(* Logix 5000 project; controller NSH_PLC1 vendor 1 type 14 code 167 rev 32.11; software revision 32.02; part 7 of 12 *)
(* tags used below, declared in another part *)
   TempMotor : Motor;   // Temp Motor Tag for Subroutines
   H32D : Motor;   // Shr.Roll.
   H33A : Motor;   // Aspirator
   H34A : Motor;   // HC Vib.
   H34B : Motor;   // Hard Crkr.
   H34C : Motor;   // S.Roll
   H34D : Motor;   // Shr.Roll.
   H35A : Motor;   // Aspirator
   H35B : Motor;   // Aspirator
   H42A : Motor;   // HC Vib.
   H42B : Motor;   // Hard Crkr.
   H42C : Motor;   // S.Roll
   H42D : Motor;   // Shr.Roll.
   H43A : Motor;   // Aspirator
   H43B : Motor;   // Aspirator
   H44A : Motor;   // HC Vib.
   H44B : Motor;   // Hard Crkr.
   H44C : Motor;   // S.Roll
   H44D : Motor;   // Shr.Roll.
   H45A : Motor;   // Aspirator
   H45B : Motor;   // Aspirator
   H49 : Motor;   // Ele.
   H50A : Motor;   // Auger
   H50B : Motor;   // Auger
   M10 : Motor;   // Vib.
   M10A : Motor;   // Asp.
   M10B : Motor;   // Asp.
   M11 : Motor;   // Ele.
   M16 : Motor;   // Evo.
   M17 : Motor;   // Evo.
   M18 : Motor;   // Vib.
   M19 : Motor;   // Ele.
   M1A : Motor;   // Vib.
   M2 : Motor;   // Vib.
   M27 : Motor;   // Belt
   M28 : Motor;   // Belt
   M29 : Motor;   // Ele.
   M3 : Motor;   // Belt
   M30A : Motor;   // HC Vib.
   M30B : Motor;   // Hard Crkr.
   M30C : Motor;   // Shr.Roll.
   M30D : Motor;   // Shr.Roll.
   M31A : Motor;   // Asp.
   M31B : Motor;   // Asp.
   M32A : Motor;   // Vib.Scrn.
   M32B : Motor;   // Ele.
   M37 : Motor;   // 5x12
   M38A : Motor;   // Asp.
   M38B : Motor;   // Asp.
   M39 : Motor;   // Ele.
   M4 : Motor;   // Vib.
   M40A : Motor;   // Sep.
   M40B : Motor;   // Syn.Fer.
   M41 : Motor;   // Ele.
   M44A : Motor;   // Belt
   M44B : Motor;   // Belt
   M5 : Motor;   // Vib.
   M6 : Motor;   // Belt
   M7 : Motor;   // Ele.
   M8 : Motor;   // Shkr.
   M9A : Motor;   // Asp.
   M9B : Motor;   // Asp.
   S1 : Motor;   // Vib.
   S10 : Motor;   // Auger
   S13 : Motor;   // Ele.
   S14 : Motor;   // Auger
   S15 : Motor;   // Auger
   S16A : Motor;   // Auger
   S16B : Motor;   // Auger
   S17A : Motor;   // HS Cracker
   S17B : Motor;   // Hard Crkr.
   S17C : Motor;   // Shr.Roll.
   S17D : Motor;   // S.Roll
   S18A : Motor;   // HC Vib.
   S18B : Motor;   // Hard Crkr.
   S18C : Motor;   // Shr.Roll.
   S18D : Motor;   // S.Roll
   S19 : Motor;   // Gry.
   S2 : Motor;   // Ele.
   S20 : Motor;   // Ele.
   S21 : Motor;   // Roll Fdr.
   S22A : Motor;   // HC Vib.
   S22B : Motor;   // Hard Crkr.
   S22C : Motor;   // Shr.Roll.
   S22D : Motor;   // S.Roll
   S23A : Motor;   // HC Vib.
   S23B : Motor;   // Hard Crkr.
   S23C : Motor;   // Shr.Roll.
   S23D : Motor;   // S.Roll
   S24 : Motor;   // Deck
   S25 : Motor;   // Ele.
   S26 : Motor;   // Auger
   S27 : Motor;   // Roll Fdr
   S28A : Motor;   // HC Vib.
   S28B : Motor;   // Hard Crkr.
   S28C : Motor;   // Shr.Roll.
   S28D : Motor;   // S.Roll
   S29A : Motor;   // HC Vib.
   S29B : Motor;   // Hard Crkr.
   S29C : Motor;   // Shr.Roll.
   S29D : Motor;   // S.Roll
   S3 : Motor;   // Auger
   S30 : Motor;   // Ele.
   S31 : Motor;   // Auger
   S32A : Motor;   // HC Vib.
   S32B : Motor;   // Hard Crkr.
   S32C : Motor;   // Shr.Roll.
   S32D : Motor;   // S.Roll
   S33A : Motor;   // HC Vib.
   S33B : Motor;   // Hard Crkr.
   S33C : Motor;   // Shr.Roll.
   S33D : Motor;   // S.Roll
   S34 : Motor;   // Deck
   S35 : Motor;   // Ele.
   S36 : Motor;   // Auger
   S37A : Motor;   // HC Vib.
   S37B : Motor;   // Hard Crkr.
   S37C : Motor;   // Shr.Roll.
   S37D : Motor;   // S.Roll
   S38 : Motor;   // Shkr.
   S39 : Motor;   // Ele.
   S40A : Motor;   // HC Vib.
   S40B : Motor;   // Hard Crkr.
   S40C : Motor;   // Shr.Roll.
   S40D : Motor;   // S.Roll
   S41 : Motor;   // Ele.
   S42A : Motor;   // HC Vib.
   S42B : Motor;   // Hard Crkr.
   S42C : Motor;   // S.Roll
   S42D : Motor;   // Shr.Roll.
   S43 : Motor;   // Shkr.
   S44 : Motor;   // Ele.
   S45 : Motor;   // Auger
   S46A : Motor;   // HC Vib.
   S46B : Motor;   // Hard Crkr.
   S46C : Motor;   // S.Roll
   S46D : Motor;   // Shr.Roll.
   S4A : Motor;   // Aspirator
   S4B : Motor;   // Aspirator
   S5A : Motor;   // Aspirator
   S5B : Motor;   // Aspirator
   S6 : Motor;   // Belt
   S7 : Motor;   // Ele.
   S8 : Motor;   // Auger
   S9 : Motor;   // Ele.
(* HullerSheller, continued *)

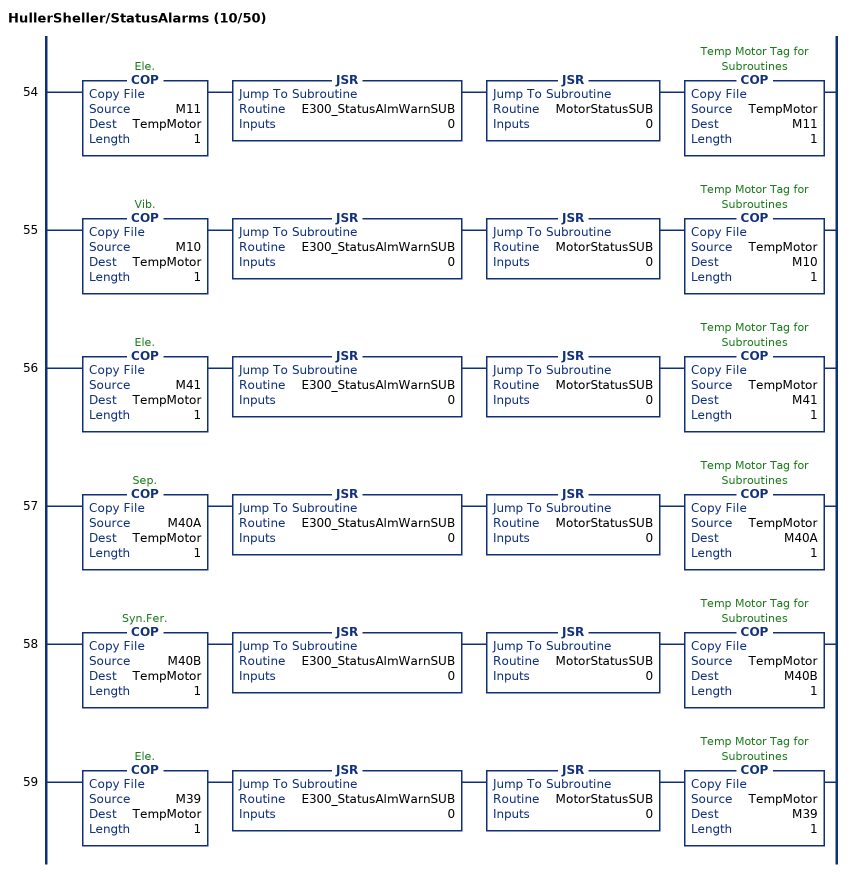
   [picture p138: HullerSheller/StatusAlarms rungs 54-59]
   54: COP(M11,TempMotor,1)JSR(E300_StatusAlmWarnSUB,0)JSR(MotorStatusSUB,0)COP(TempMotor,M11,1);
   55: COP(M10,TempMotor,1)JSR(E300_StatusAlmWarnSUB,0)JSR(MotorStatusSUB,0)COP(TempMotor,M10,1);
   56: COP(M41,TempMotor,1)JSR(E300_StatusAlmWarnSUB,0)JSR(MotorStatusSUB,0)COP(TempMotor,M41,1);
   57: COP(M40A,TempMotor,1)JSR(E300_StatusAlmWarnSUB,0)JSR(MotorStatusSUB,0)COP(TempMotor,M40A,1);
   58: COP(M40B,TempMotor,1)JSR(E300_StatusAlmWarnSUB,0)JSR(MotorStatusSUB,0)COP(TempMotor,M40B,1);
   59: COP(M39,TempMotor,1)JSR(E300_StatusAlmWarnSUB,0)JSR(MotorStatusSUB,0)COP(TempMotor,M39,1);
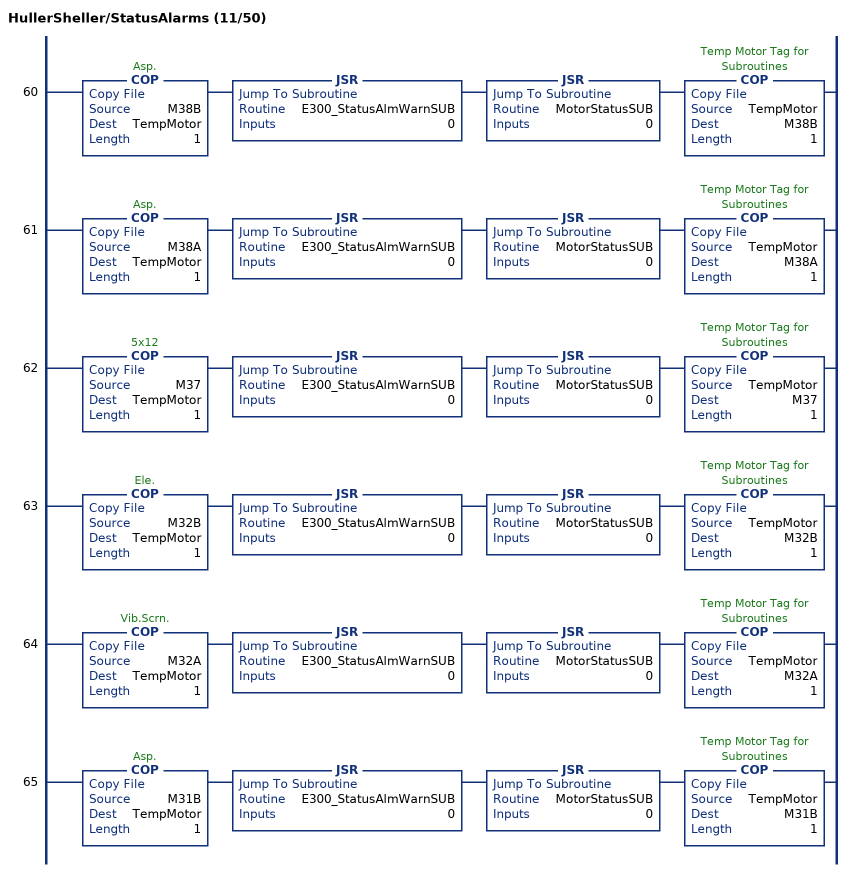
   60: COP(M38B,TempMotor,1)JSR(E300_StatusAlmWarnSUB,0)JSR(MotorStatusSUB,0)COP(TempMotor,M38B,1);
   61: COP(M38A,TempMotor,1)JSR(E300_StatusAlmWarnSUB,0)JSR(MotorStatusSUB,0)COP(TempMotor,M38A,1);
   62: COP(M37,TempMotor,1)JSR(E300_StatusAlmWarnSUB,0)JSR(MotorStatusSUB,0)COP(TempMotor,M37,1);
   63: COP(M32B,TempMotor,1)JSR(E300_StatusAlmWarnSUB,0)JSR(MotorStatusSUB,0)COP(TempMotor,M32B,1);
   64: COP(M32A,TempMotor,1)JSR(E300_StatusAlmWarnSUB,0)JSR(MotorStatusSUB,0)COP(TempMotor,M32A,1);
   65: COP(M31B,TempMotor,1)JSR(E300_StatusAlmWarnSUB,0)JSR(MotorStatusSUB,0)COP(TempMotor,M31B,1);
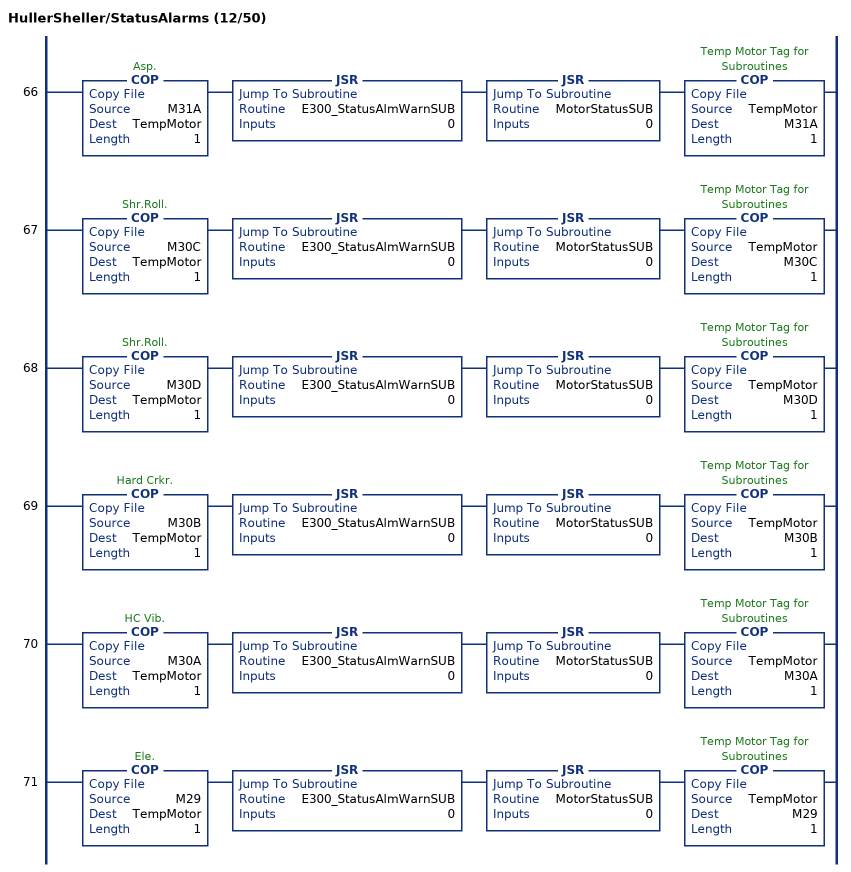
   66: COP(M31A,TempMotor,1)JSR(E300_StatusAlmWarnSUB,0)JSR(MotorStatusSUB,0)COP(TempMotor,M31A,1);
   67: COP(M30C,TempMotor,1)JSR(E300_StatusAlmWarnSUB,0)JSR(MotorStatusSUB,0)COP(TempMotor,M30C,1);
   68: COP(M30D,TempMotor,1)JSR(E300_StatusAlmWarnSUB,0)JSR(MotorStatusSUB,0)COP(TempMotor,M30D,1);
   69: COP(M30B,TempMotor,1)JSR(E300_StatusAlmWarnSUB,0)JSR(MotorStatusSUB,0)COP(TempMotor,M30B,1);
   70: COP(M30A,TempMotor,1)JSR(E300_StatusAlmWarnSUB,0)JSR(MotorStatusSUB,0)COP(TempMotor,M30A,1);
   71: COP(M29,TempMotor,1)JSR(E300_StatusAlmWarnSUB,0)JSR(MotorStatusSUB,0)COP(TempMotor,M29,1);
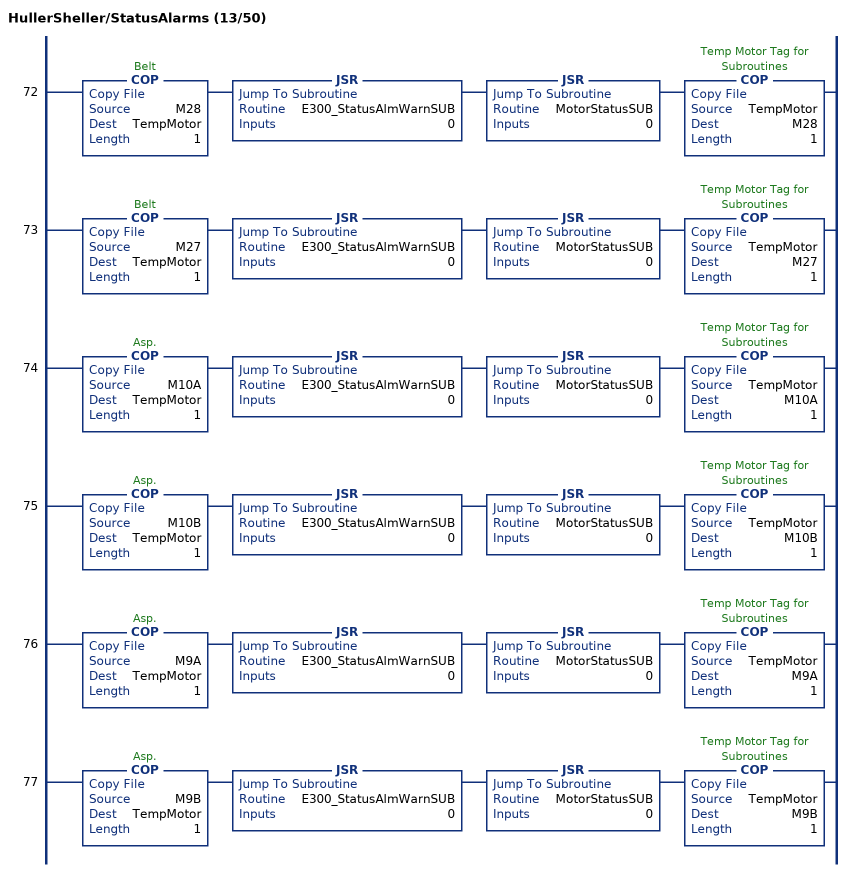
   72: COP(M28,TempMotor,1)JSR(E300_StatusAlmWarnSUB,0)JSR(MotorStatusSUB,0)COP(TempMotor,M28,1);
   73: COP(M27,TempMotor,1)JSR(E300_StatusAlmWarnSUB,0)JSR(MotorStatusSUB,0)COP(TempMotor,M27,1);
   74: COP(M10A,TempMotor,1)JSR(E300_StatusAlmWarnSUB,0)JSR(MotorStatusSUB,0)COP(TempMotor,M10A,1);
   75: COP(M10B,TempMotor,1)JSR(E300_StatusAlmWarnSUB,0)JSR(MotorStatusSUB,0)COP(TempMotor,M10B,1);
   76: COP(M9A,TempMotor,1)JSR(E300_StatusAlmWarnSUB,0)JSR(MotorStatusSUB,0)COP(TempMotor,M9A,1);
   77: COP(M9B,TempMotor,1)JSR(E300_StatusAlmWarnSUB,0)JSR(MotorStatusSUB,0)COP(TempMotor,M9B,1);
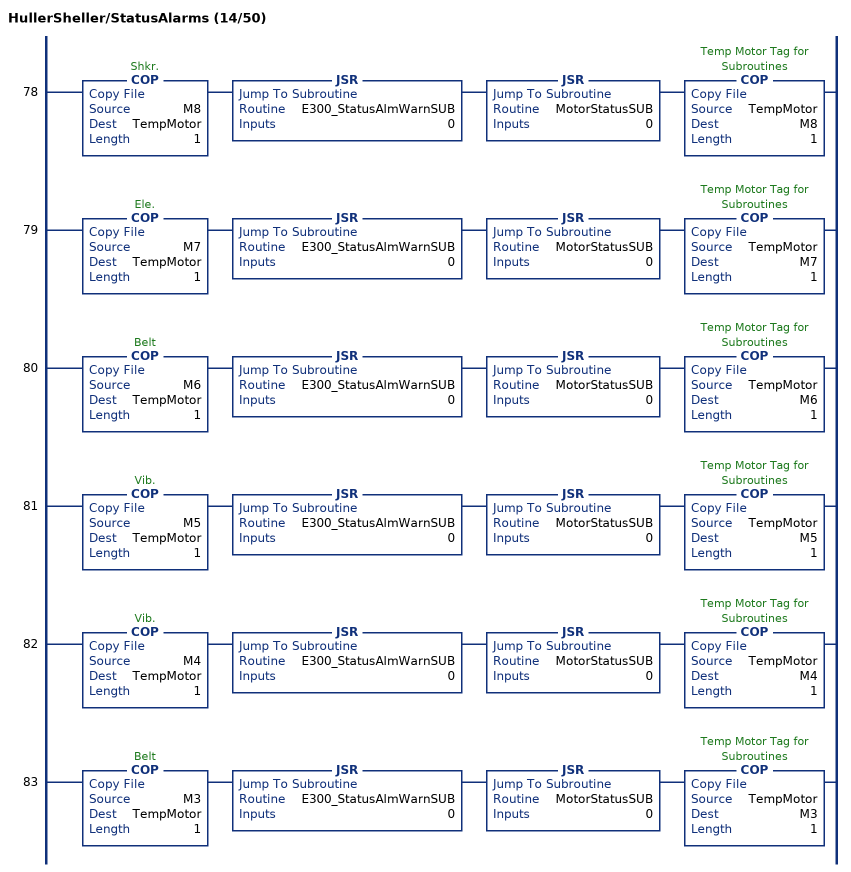
   78: COP(M8,TempMotor,1)JSR(E300_StatusAlmWarnSUB,0)JSR(MotorStatusSUB,0)COP(TempMotor,M8,1);
   79: COP(M7,TempMotor,1)JSR(E300_StatusAlmWarnSUB,0)JSR(MotorStatusSUB,0)COP(TempMotor,M7,1);
   80: COP(M6,TempMotor,1)JSR(E300_StatusAlmWarnSUB,0)JSR(MotorStatusSUB,0)COP(TempMotor,M6,1);
   81: COP(M5,TempMotor,1)JSR(E300_StatusAlmWarnSUB,0)JSR(MotorStatusSUB,0)COP(TempMotor,M5,1);
   82: COP(M4,TempMotor,1)JSR(E300_StatusAlmWarnSUB,0)JSR(MotorStatusSUB,0)COP(TempMotor,M4,1);
   83: COP(M3,TempMotor,1)JSR(E300_StatusAlmWarnSUB,0)JSR(MotorStatusSUB,0)COP(TempMotor,M3,1);
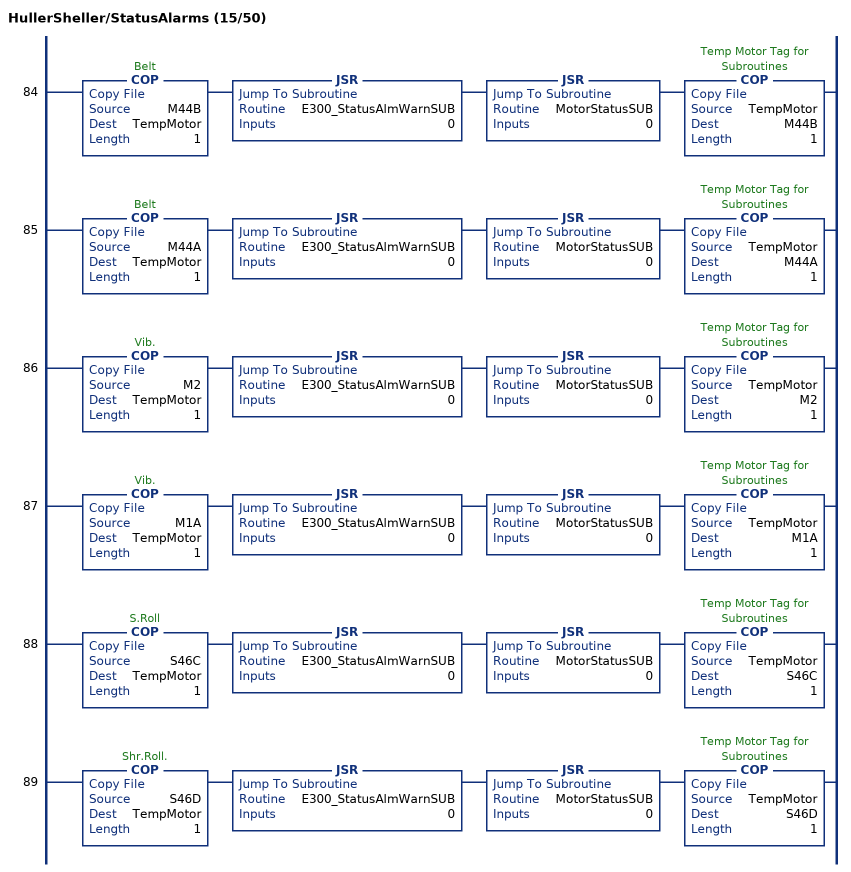
   84: COP(M44B,TempMotor,1)JSR(E300_StatusAlmWarnSUB,0)JSR(MotorStatusSUB,0)COP(TempMotor,M44B,1);
   85: COP(M44A,TempMotor,1)JSR(E300_StatusAlmWarnSUB,0)JSR(MotorStatusSUB,0)COP(TempMotor,M44A,1);
   86: COP(M2,TempMotor,1)JSR(E300_StatusAlmWarnSUB,0)JSR(MotorStatusSUB,0)COP(TempMotor,M2,1);
   87: COP(M1A,TempMotor,1)JSR(E300_StatusAlmWarnSUB,0)JSR(MotorStatusSUB,0)COP(TempMotor,M1A,1);
   88: COP(S46C,TempMotor,1)JSR(E300_StatusAlmWarnSUB,0)JSR(MotorStatusSUB,0)COP(TempMotor,S46C,1);
   89: COP(S46D,TempMotor,1)JSR(E300_StatusAlmWarnSUB,0)JSR(MotorStatusSUB,0)COP(TempMotor,S46D,1);
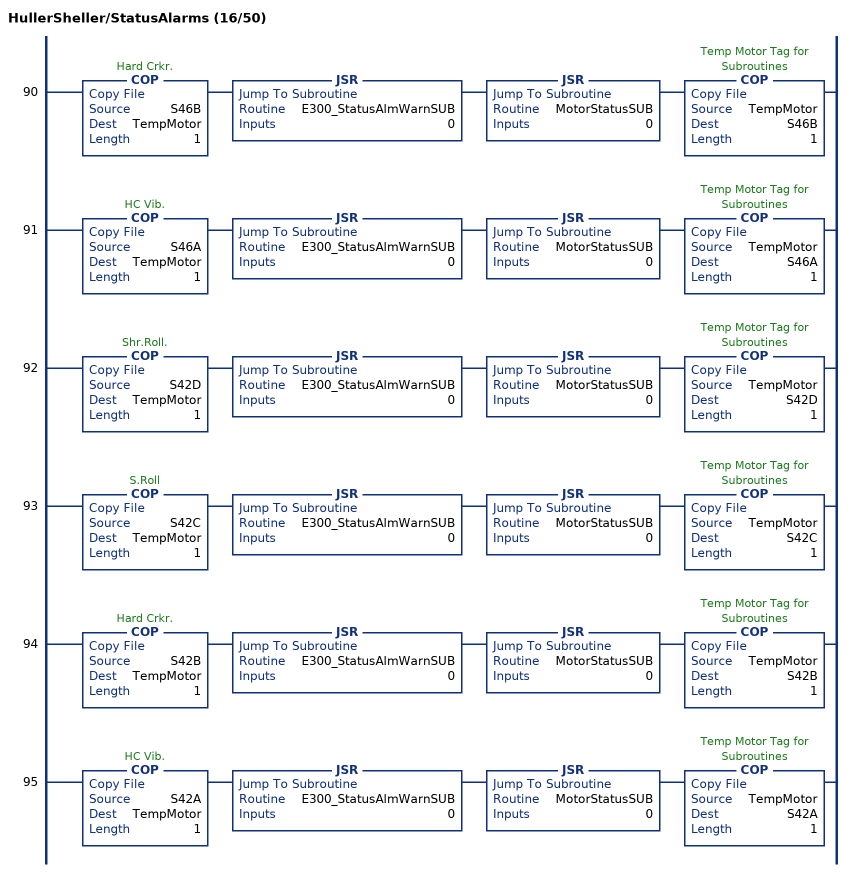
   90: COP(S46B,TempMotor,1)JSR(E300_StatusAlmWarnSUB,0)JSR(MotorStatusSUB,0)COP(TempMotor,S46B,1);
   91: COP(S46A,TempMotor,1)JSR(E300_StatusAlmWarnSUB,0)JSR(MotorStatusSUB,0)COP(TempMotor,S46A,1);
   92: COP(S42D,TempMotor,1)JSR(E300_StatusAlmWarnSUB,0)JSR(MotorStatusSUB,0)COP(TempMotor,S42D,1);
   93: COP(S42C,TempMotor,1)JSR(E300_StatusAlmWarnSUB,0)JSR(MotorStatusSUB,0)COP(TempMotor,S42C,1);
   94: COP(S42B,TempMotor,1)JSR(E300_StatusAlmWarnSUB,0)JSR(MotorStatusSUB,0)COP(TempMotor,S42B,1);
   95: COP(S42A,TempMotor,1)JSR(E300_StatusAlmWarnSUB,0)JSR(MotorStatusSUB,0)COP(TempMotor,S42A,1);
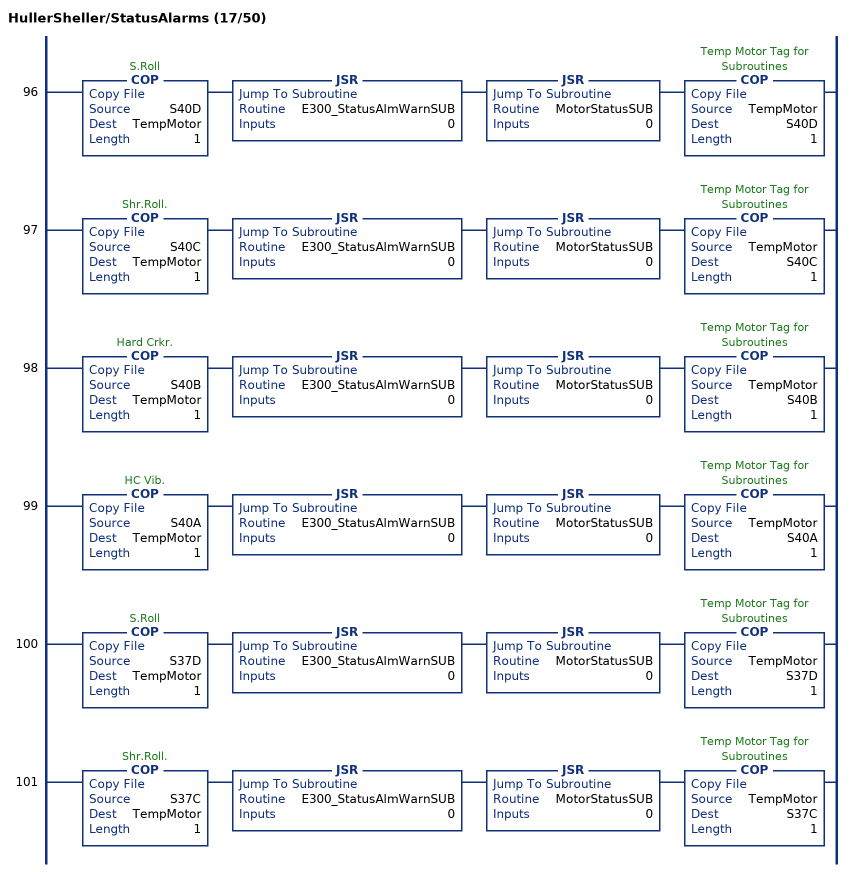
   96: COP(S40D,TempMotor,1)JSR(E300_StatusAlmWarnSUB,0)JSR(MotorStatusSUB,0)COP(TempMotor,S40D,1);
   97: COP(S40C,TempMotor,1)JSR(E300_StatusAlmWarnSUB,0)JSR(MotorStatusSUB,0)COP(TempMotor,S40C,1);
   98: COP(S40B,TempMotor,1)JSR(E300_StatusAlmWarnSUB,0)JSR(MotorStatusSUB,0)COP(TempMotor,S40B,1);
   99: COP(S40A,TempMotor,1)JSR(E300_StatusAlmWarnSUB,0)JSR(MotorStatusSUB,0)COP(TempMotor,S40A,1);
   100: COP(S37D,TempMotor,1)JSR(E300_StatusAlmWarnSUB,0)JSR(MotorStatusSUB,0)COP(TempMotor,S37D,1);
   101: COP(S37C,TempMotor,1)JSR(E300_StatusAlmWarnSUB,0)JSR(MotorStatusSUB,0)COP(TempMotor,S37C,1);
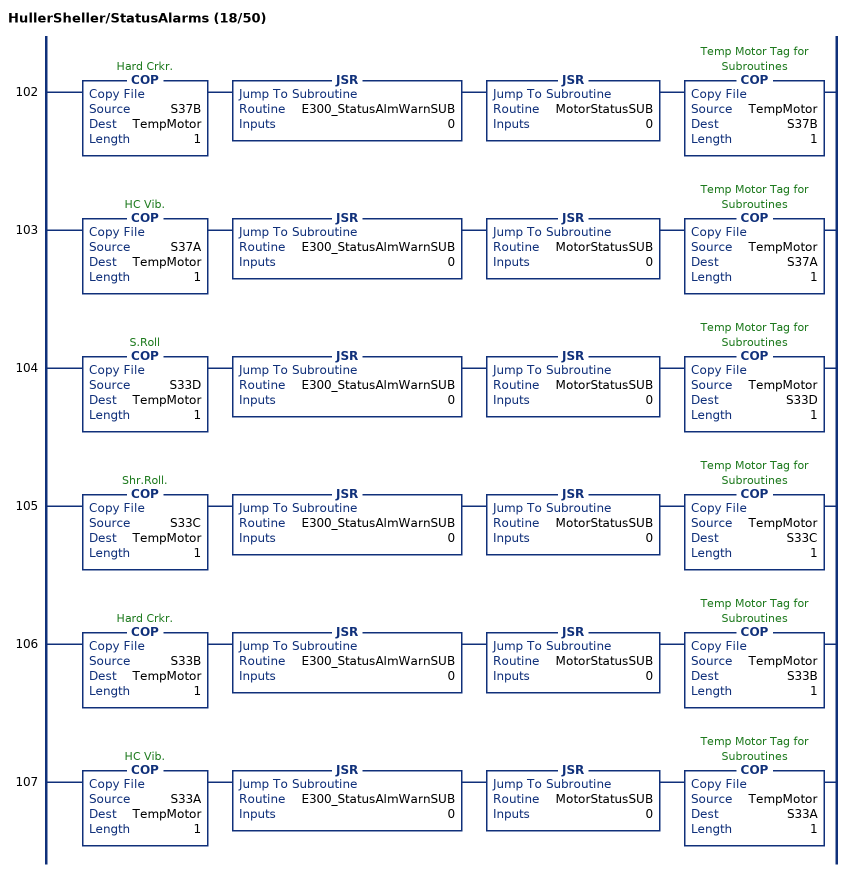
   102: COP(S37B,TempMotor,1)JSR(E300_StatusAlmWarnSUB,0)JSR(MotorStatusSUB,0)COP(TempMotor,S37B,1);
   103: COP(S37A,TempMotor,1)JSR(E300_StatusAlmWarnSUB,0)JSR(MotorStatusSUB,0)COP(TempMotor,S37A,1);
   104: COP(S33D,TempMotor,1)JSR(E300_StatusAlmWarnSUB,0)JSR(MotorStatusSUB,0)COP(TempMotor,S33D,1);
   105: COP(S33C,TempMotor,1)JSR(E300_StatusAlmWarnSUB,0)JSR(MotorStatusSUB,0)COP(TempMotor,S33C,1);
   106: COP(S33B,TempMotor,1)JSR(E300_StatusAlmWarnSUB,0)JSR(MotorStatusSUB,0)COP(TempMotor,S33B,1);
   107: COP(S33A,TempMotor,1)JSR(E300_StatusAlmWarnSUB,0)JSR(MotorStatusSUB,0)COP(TempMotor,S33A,1);
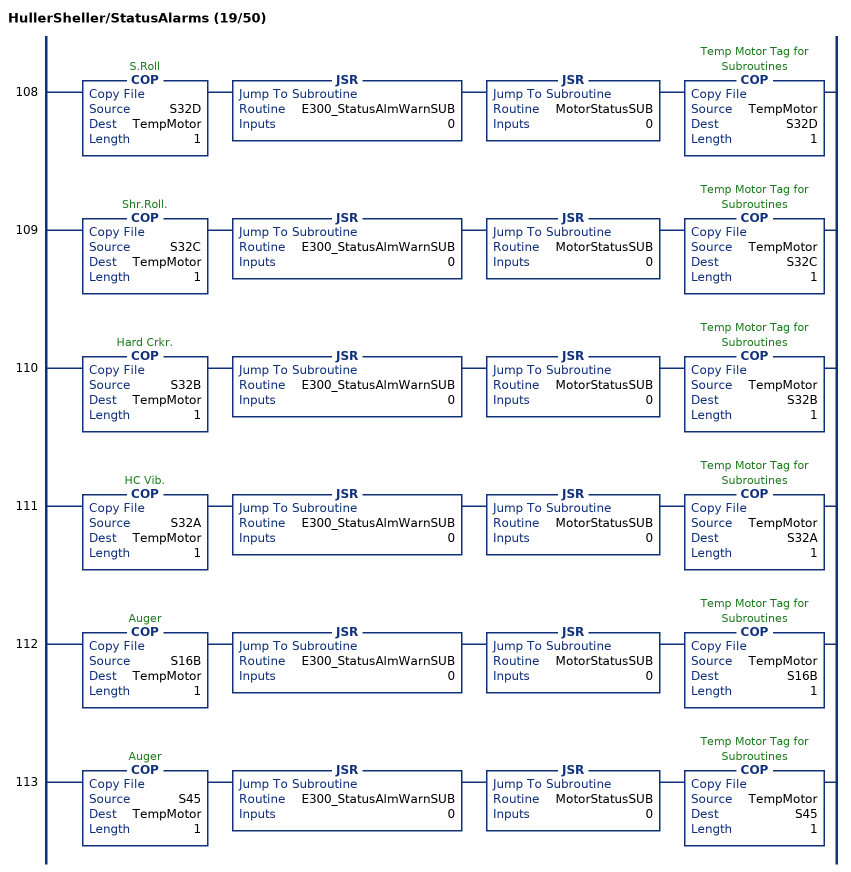
   108: COP(S32D,TempMotor,1)JSR(E300_StatusAlmWarnSUB,0)JSR(MotorStatusSUB,0)COP(TempMotor,S32D,1);
   109: COP(S32C,TempMotor,1)JSR(E300_StatusAlmWarnSUB,0)JSR(MotorStatusSUB,0)COP(TempMotor,S32C,1);
   110: COP(S32B,TempMotor,1)JSR(E300_StatusAlmWarnSUB,0)JSR(MotorStatusSUB,0)COP(TempMotor,S32B,1);
   111: COP(S32A,TempMotor,1)JSR(E300_StatusAlmWarnSUB,0)JSR(MotorStatusSUB,0)COP(TempMotor,S32A,1);
   112: COP(S16B,TempMotor,1)JSR(E300_StatusAlmWarnSUB,0)JSR(MotorStatusSUB,0)COP(TempMotor,S16B,1);
   113: COP(S45,TempMotor,1)JSR(E300_StatusAlmWarnSUB,0)JSR(MotorStatusSUB,0)COP(TempMotor,S45,1);
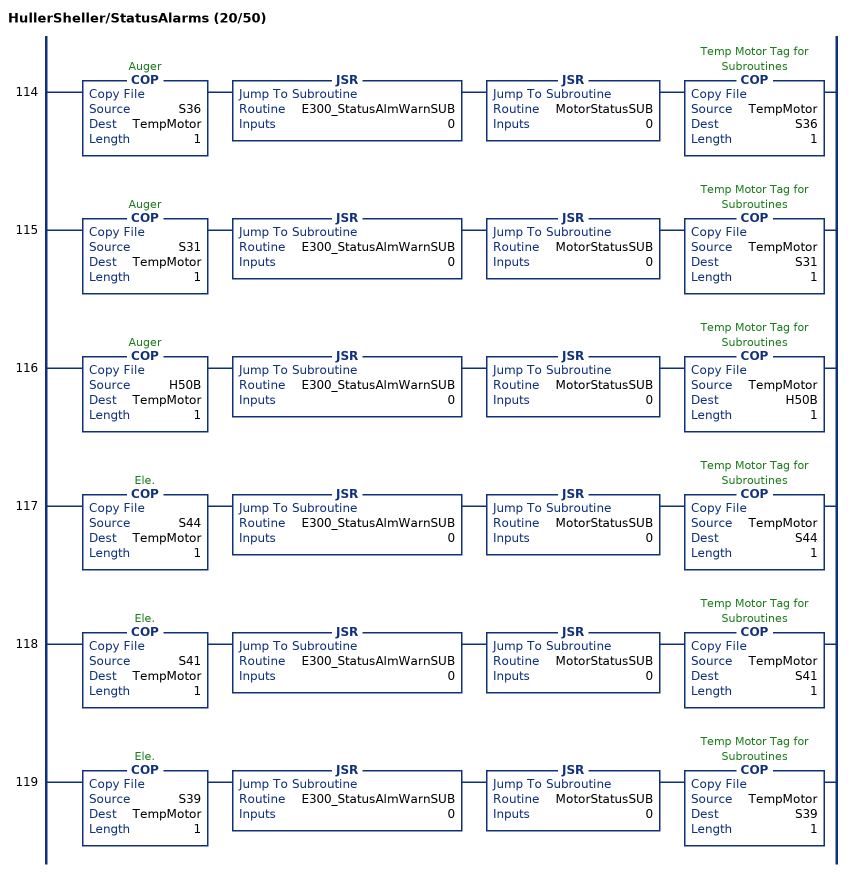
   114: COP(S36,TempMotor,1)JSR(E300_StatusAlmWarnSUB,0)JSR(MotorStatusSUB,0)COP(TempMotor,S36,1);
   115: COP(S31,TempMotor,1)JSR(E300_StatusAlmWarnSUB,0)JSR(MotorStatusSUB,0)COP(TempMotor,S31,1);
   116: COP(H50B,TempMotor,1)JSR(E300_StatusAlmWarnSUB,0)JSR(MotorStatusSUB,0)COP(TempMotor,H50B,1);
   117: COP(S44,TempMotor,1)JSR(E300_StatusAlmWarnSUB,0)JSR(MotorStatusSUB,0)COP(TempMotor,S44,1);
   118: COP(S41,TempMotor,1)JSR(E300_StatusAlmWarnSUB,0)JSR(MotorStatusSUB,0)COP(TempMotor,S41,1);
   119: COP(S39,TempMotor,1)JSR(E300_StatusAlmWarnSUB,0)JSR(MotorStatusSUB,0)COP(TempMotor,S39,1);
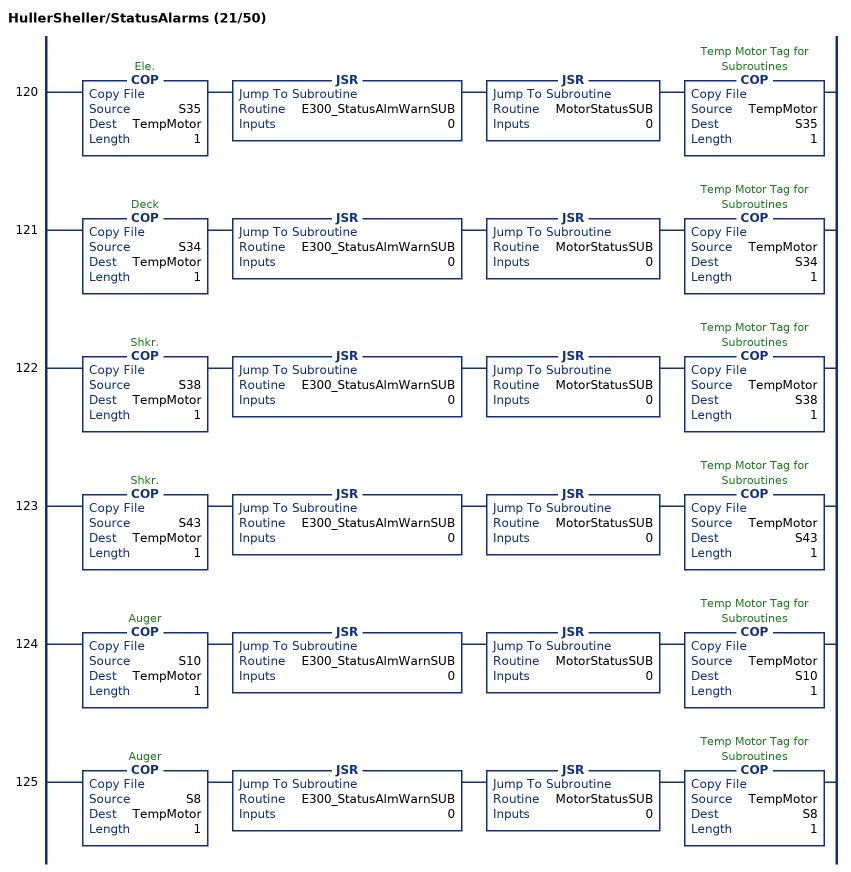
   120: COP(S35,TempMotor,1)JSR(E300_StatusAlmWarnSUB,0)JSR(MotorStatusSUB,0)COP(TempMotor,S35,1);
   121: COP(S34,TempMotor,1)JSR(E300_StatusAlmWarnSUB,0)JSR(MotorStatusSUB,0)COP(TempMotor,S34,1);
   122: COP(S38,TempMotor,1)JSR(E300_StatusAlmWarnSUB,0)JSR(MotorStatusSUB,0)COP(TempMotor,S38,1);
   123: COP(S43,TempMotor,1)JSR(E300_StatusAlmWarnSUB,0)JSR(MotorStatusSUB,0)COP(TempMotor,S43,1);
   124: COP(S10,TempMotor,1)JSR(E300_StatusAlmWarnSUB,0)JSR(MotorStatusSUB,0)COP(TempMotor,S10,1);
   125: COP(S8,TempMotor,1)JSR(E300_StatusAlmWarnSUB,0)JSR(MotorStatusSUB,0)COP(TempMotor,S8,1);
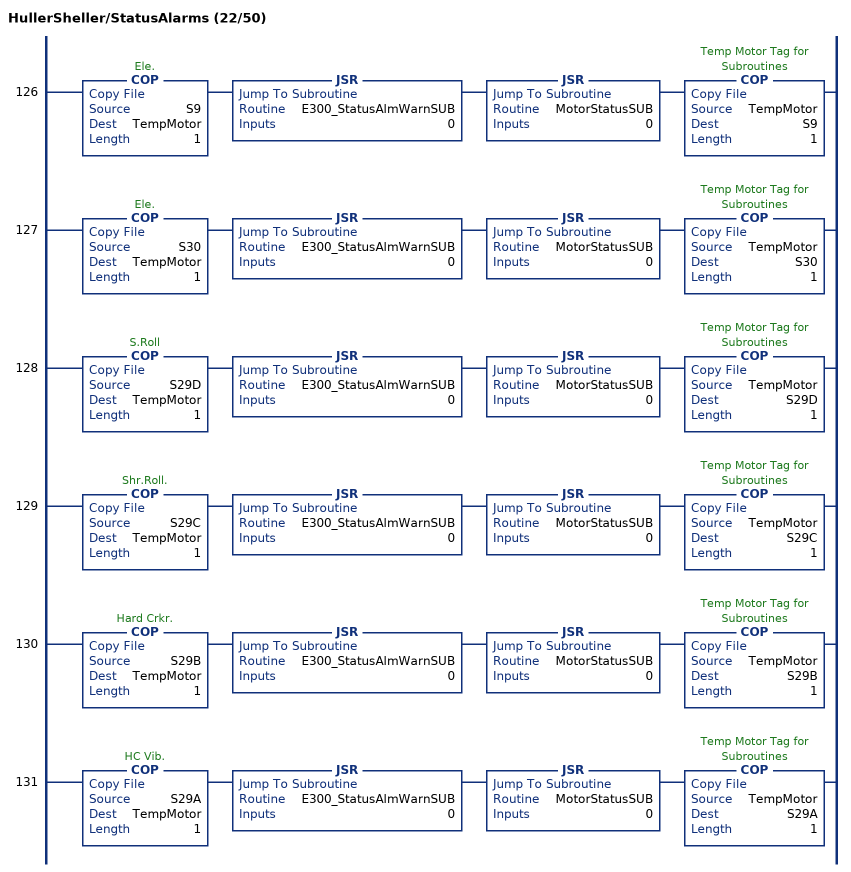
   126: COP(S9,TempMotor,1)JSR(E300_StatusAlmWarnSUB,0)JSR(MotorStatusSUB,0)COP(TempMotor,S9,1);
   127: COP(S30,TempMotor,1)JSR(E300_StatusAlmWarnSUB,0)JSR(MotorStatusSUB,0)COP(TempMotor,S30,1);
   128: COP(S29D,TempMotor,1)JSR(E300_StatusAlmWarnSUB,0)JSR(MotorStatusSUB,0)COP(TempMotor,S29D,1);
   129: COP(S29C,TempMotor,1)JSR(E300_StatusAlmWarnSUB,0)JSR(MotorStatusSUB,0)COP(TempMotor,S29C,1);
   130: COP(S29B,TempMotor,1)JSR(E300_StatusAlmWarnSUB,0)JSR(MotorStatusSUB,0)COP(TempMotor,S29B,1);
   131: COP(S29A,TempMotor,1)JSR(E300_StatusAlmWarnSUB,0)JSR(MotorStatusSUB,0)COP(TempMotor,S29A,1);
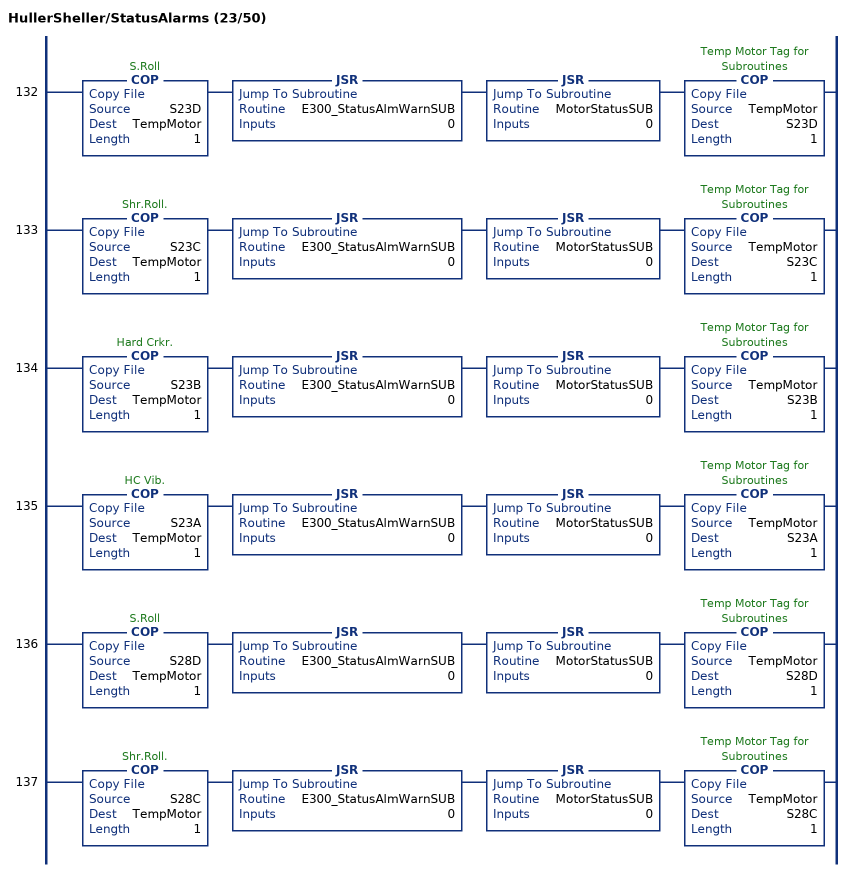
   132: COP(S23D,TempMotor,1)JSR(E300_StatusAlmWarnSUB,0)JSR(MotorStatusSUB,0)COP(TempMotor,S23D,1);
   133: COP(S23C,TempMotor,1)JSR(E300_StatusAlmWarnSUB,0)JSR(MotorStatusSUB,0)COP(TempMotor,S23C,1);
   134: COP(S23B,TempMotor,1)JSR(E300_StatusAlmWarnSUB,0)JSR(MotorStatusSUB,0)COP(TempMotor,S23B,1);
   135: COP(S23A,TempMotor,1)JSR(E300_StatusAlmWarnSUB,0)JSR(MotorStatusSUB,0)COP(TempMotor,S23A,1);
   136: COP(S28D,TempMotor,1)JSR(E300_StatusAlmWarnSUB,0)JSR(MotorStatusSUB,0)COP(TempMotor,S28D,1);
   137: COP(S28C,TempMotor,1)JSR(E300_StatusAlmWarnSUB,0)JSR(MotorStatusSUB,0)COP(TempMotor,S28C,1);
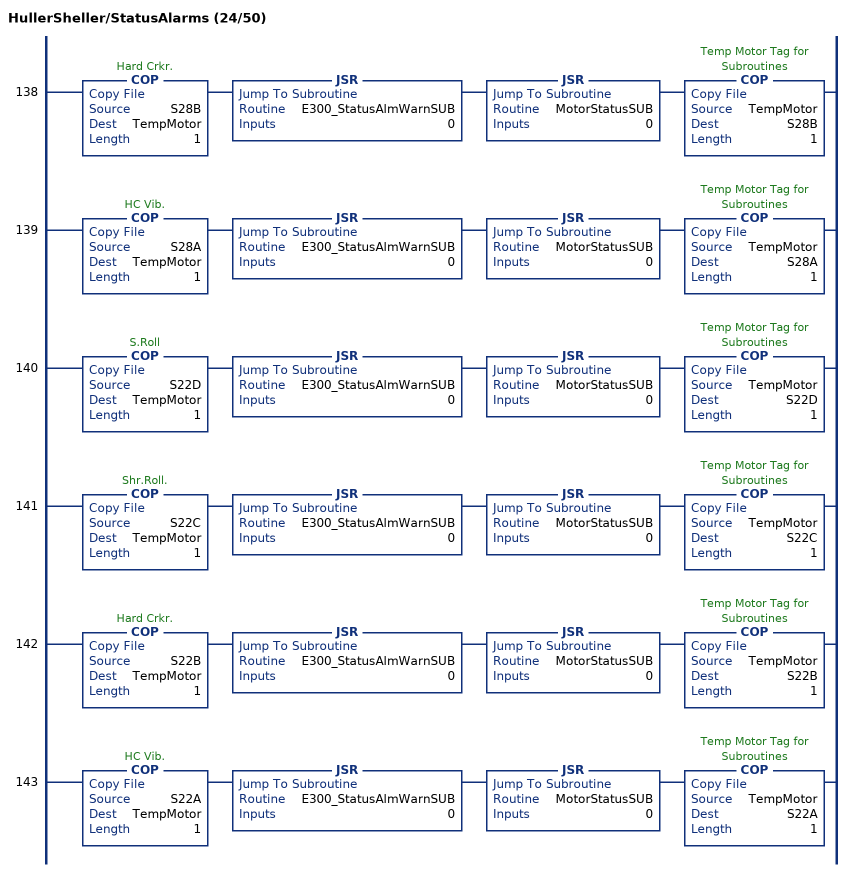
   138: COP(S28B,TempMotor,1)JSR(E300_StatusAlmWarnSUB,0)JSR(MotorStatusSUB,0)COP(TempMotor,S28B,1);
   139: COP(S28A,TempMotor,1)JSR(E300_StatusAlmWarnSUB,0)JSR(MotorStatusSUB,0)COP(TempMotor,S28A,1);
   140: COP(S22D,TempMotor,1)JSR(E300_StatusAlmWarnSUB,0)JSR(MotorStatusSUB,0)COP(TempMotor,S22D,1);
   141: COP(S22C,TempMotor,1)JSR(E300_StatusAlmWarnSUB,0)JSR(MotorStatusSUB,0)COP(TempMotor,S22C,1);
   142: COP(S22B,TempMotor,1)JSR(E300_StatusAlmWarnSUB,0)JSR(MotorStatusSUB,0)COP(TempMotor,S22B,1);
   143: COP(S22A,TempMotor,1)JSR(E300_StatusAlmWarnSUB,0)JSR(MotorStatusSUB,0)COP(TempMotor,S22A,1);
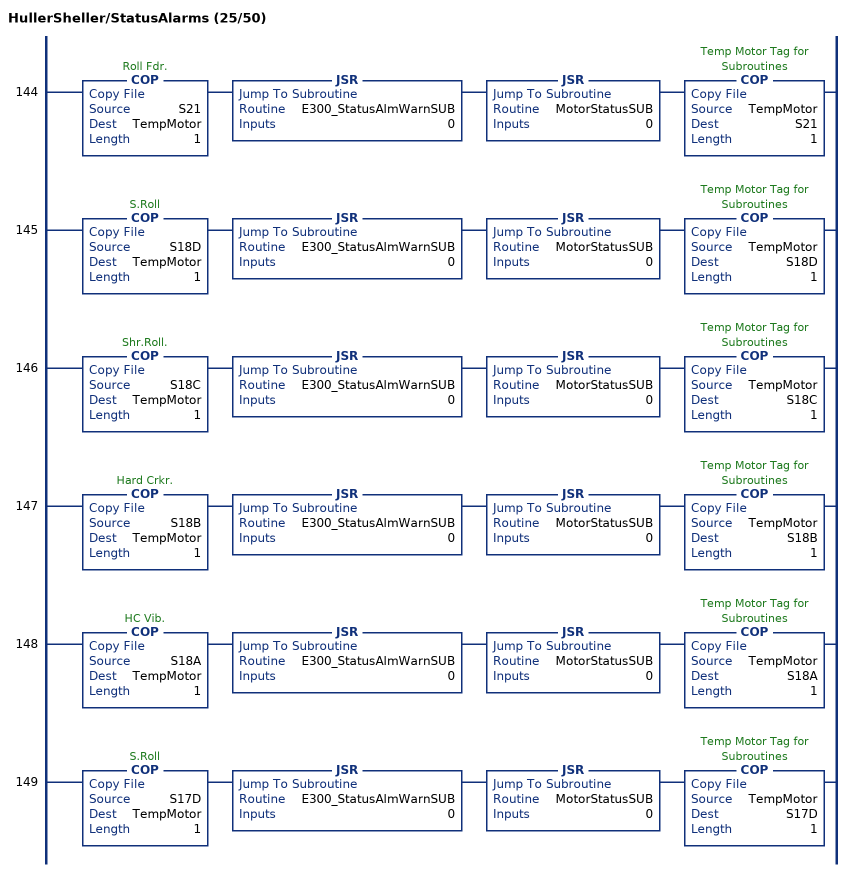
   144: COP(S21,TempMotor,1)JSR(E300_StatusAlmWarnSUB,0)JSR(MotorStatusSUB,0)COP(TempMotor,S21,1);
   145: COP(S18D,TempMotor,1)JSR(E300_StatusAlmWarnSUB,0)JSR(MotorStatusSUB,0)COP(TempMotor,S18D,1);
   146: COP(S18C,TempMotor,1)JSR(E300_StatusAlmWarnSUB,0)JSR(MotorStatusSUB,0)COP(TempMotor,S18C,1);
   147: COP(S18B,TempMotor,1)JSR(E300_StatusAlmWarnSUB,0)JSR(MotorStatusSUB,0)COP(TempMotor,S18B,1);
   148: COP(S18A,TempMotor,1)JSR(E300_StatusAlmWarnSUB,0)JSR(MotorStatusSUB,0)COP(TempMotor,S18A,1);
   149: COP(S17D,TempMotor,1)JSR(E300_StatusAlmWarnSUB,0)JSR(MotorStatusSUB,0)COP(TempMotor,S17D,1);
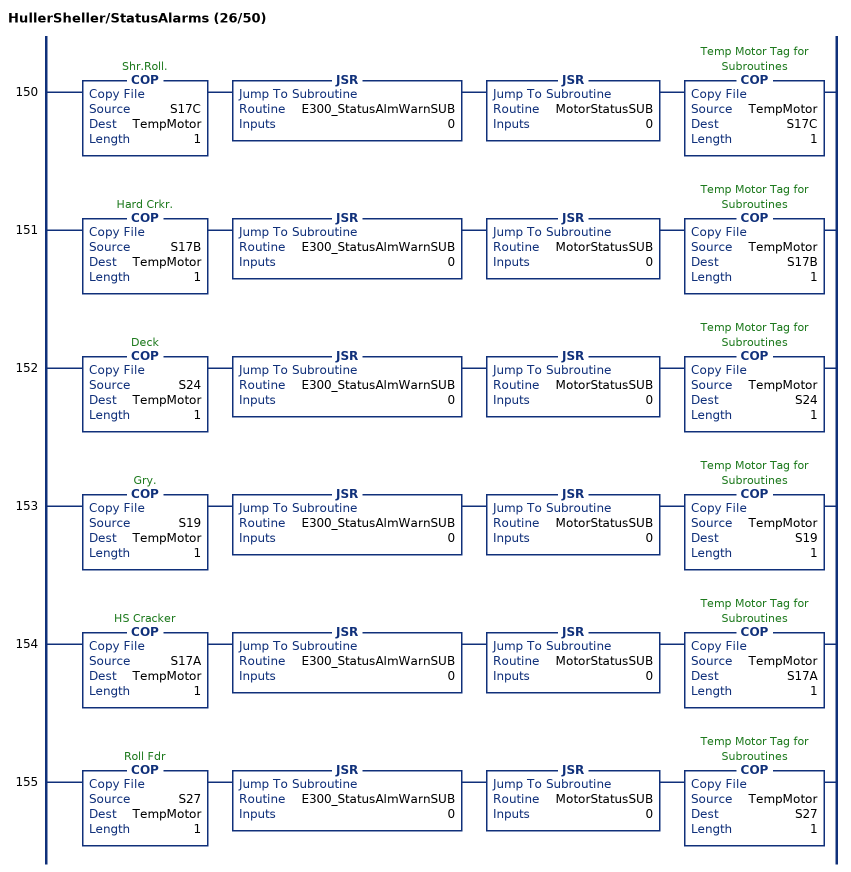
   150: COP(S17C,TempMotor,1)JSR(E300_StatusAlmWarnSUB,0)JSR(MotorStatusSUB,0)COP(TempMotor,S17C,1);
   151: COP(S17B,TempMotor,1)JSR(E300_StatusAlmWarnSUB,0)JSR(MotorStatusSUB,0)COP(TempMotor,S17B,1);
   152: COP(S24,TempMotor,1)JSR(E300_StatusAlmWarnSUB,0)JSR(MotorStatusSUB,0)COP(TempMotor,S24,1);
   153: COP(S19,TempMotor,1)JSR(E300_StatusAlmWarnSUB,0)JSR(MotorStatusSUB,0)COP(TempMotor,S19,1);
   154: COP(S17A,TempMotor,1)JSR(E300_StatusAlmWarnSUB,0)JSR(MotorStatusSUB,0)COP(TempMotor,S17A,1);
   155: COP(S27,TempMotor,1)JSR(E300_StatusAlmWarnSUB,0)JSR(MotorStatusSUB,0)COP(TempMotor,S27,1);
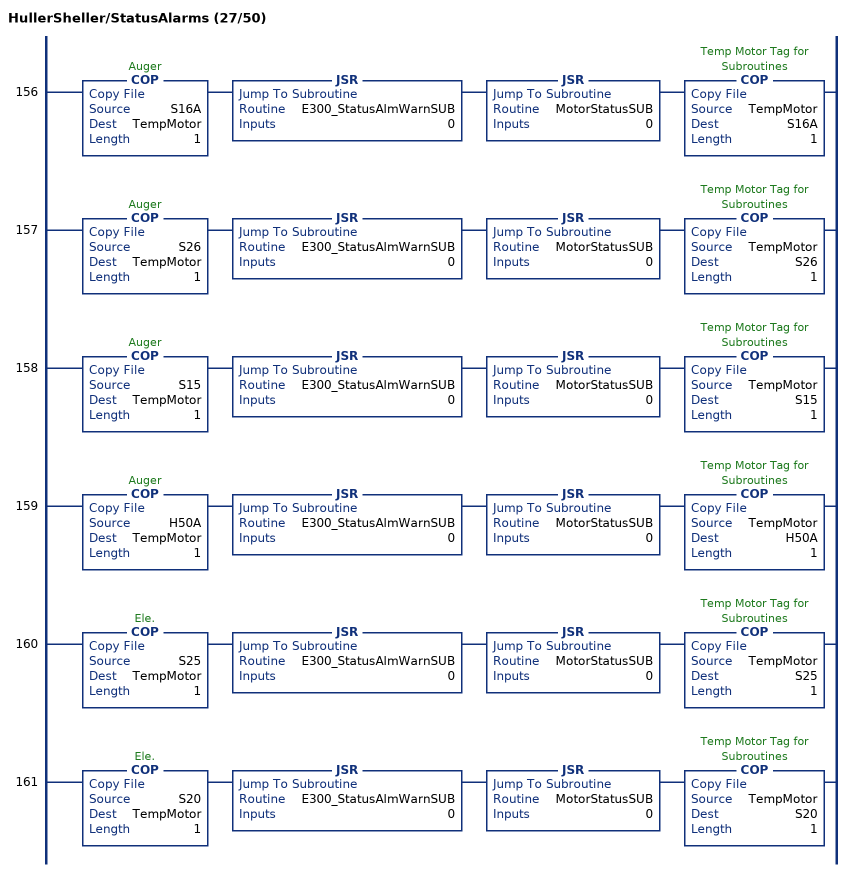
   156: COP(S16A,TempMotor,1)JSR(E300_StatusAlmWarnSUB,0)JSR(MotorStatusSUB,0)COP(TempMotor,S16A,1);
   157: COP(S26,TempMotor,1)JSR(E300_StatusAlmWarnSUB,0)JSR(MotorStatusSUB,0)COP(TempMotor,S26,1);
   158: COP(S15,TempMotor,1)JSR(E300_StatusAlmWarnSUB,0)JSR(MotorStatusSUB,0)COP(TempMotor,S15,1);
   159: COP(H50A,TempMotor,1)JSR(E300_StatusAlmWarnSUB,0)JSR(MotorStatusSUB,0)COP(TempMotor,H50A,1);
   160: COP(S25,TempMotor,1)JSR(E300_StatusAlmWarnSUB,0)JSR(MotorStatusSUB,0)COP(TempMotor,S25,1);
   161: COP(S20,TempMotor,1)JSR(E300_StatusAlmWarnSUB,0)JSR(MotorStatusSUB,0)COP(TempMotor,S20,1);
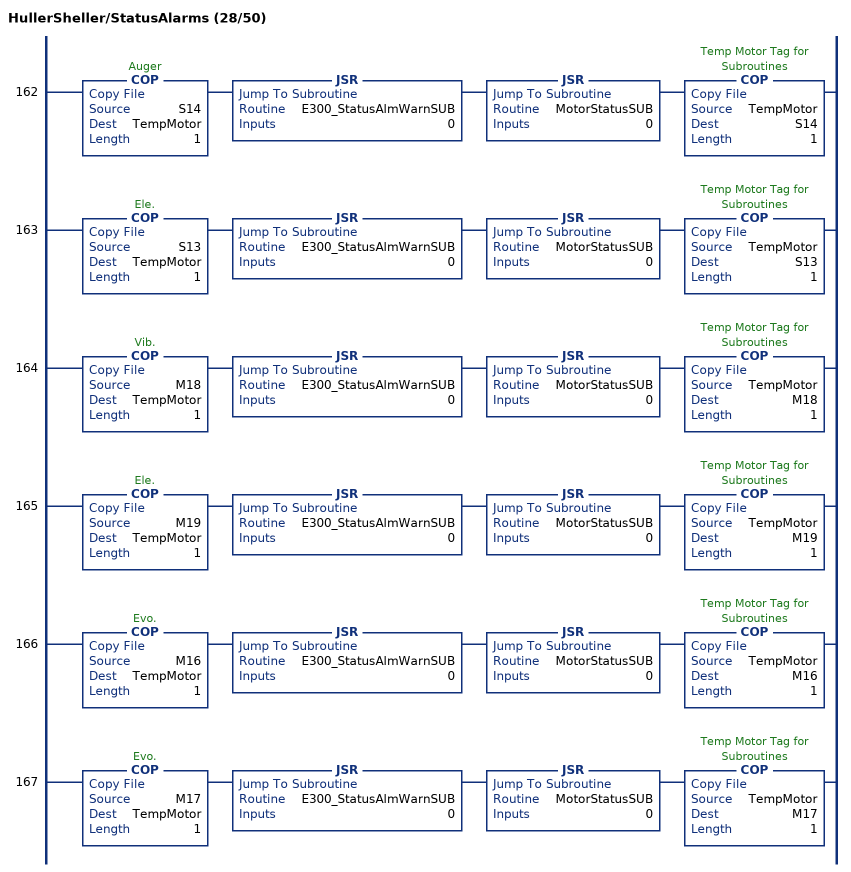
   162: COP(S14,TempMotor,1)JSR(E300_StatusAlmWarnSUB,0)JSR(MotorStatusSUB,0)COP(TempMotor,S14,1);
   163: COP(S13,TempMotor,1)JSR(E300_StatusAlmWarnSUB,0)JSR(MotorStatusSUB,0)COP(TempMotor,S13,1);
   164: COP(M18,TempMotor,1)JSR(E300_StatusAlmWarnSUB,0)JSR(MotorStatusSUB,0)COP(TempMotor,M18,1);
   165: COP(M19,TempMotor,1)JSR(E300_StatusAlmWarnSUB,0)JSR(MotorStatusSUB,0)COP(TempMotor,M19,1);
   166: COP(M16,TempMotor,1)JSR(E300_StatusAlmWarnSUB,0)JSR(MotorStatusSUB,0)COP(TempMotor,M16,1);
   167: COP(M17,TempMotor,1)JSR(E300_StatusAlmWarnSUB,0)JSR(MotorStatusSUB,0)COP(TempMotor,M17,1);
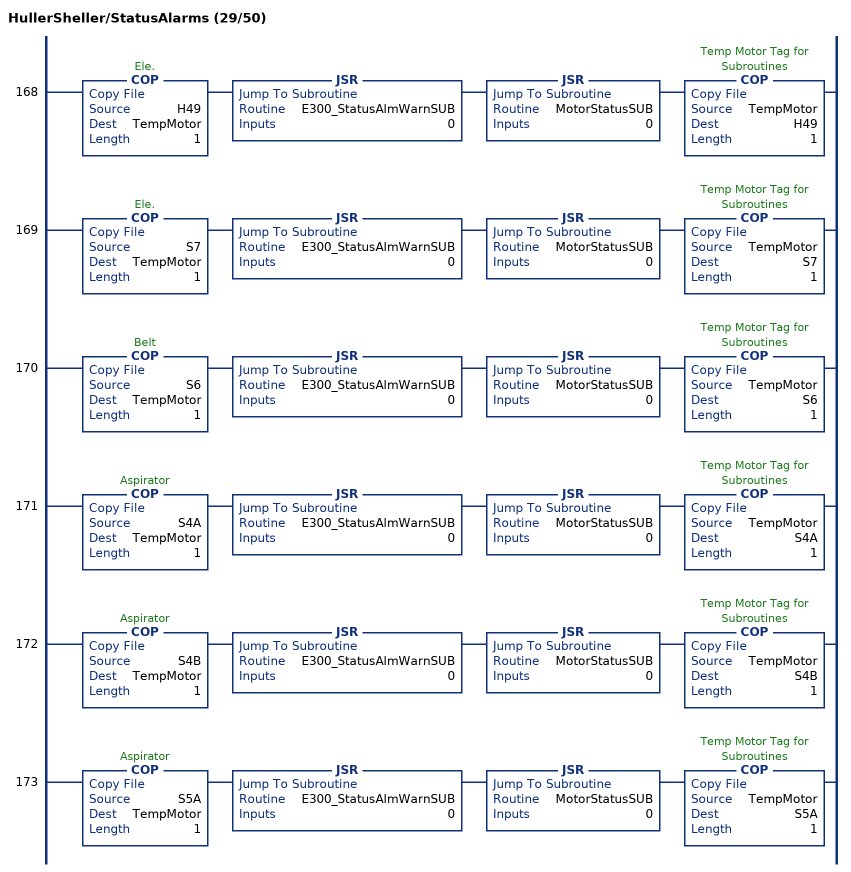
   168: COP(H49,TempMotor,1)JSR(E300_StatusAlmWarnSUB,0)JSR(MotorStatusSUB,0)COP(TempMotor,H49,1);
   169: COP(S7,TempMotor,1)JSR(E300_StatusAlmWarnSUB,0)JSR(MotorStatusSUB,0)COP(TempMotor,S7,1);
   170: COP(S6,TempMotor,1)JSR(E300_StatusAlmWarnSUB,0)JSR(MotorStatusSUB,0)COP(TempMotor,S6,1);
   171: COP(S4A,TempMotor,1)JSR(E300_StatusAlmWarnSUB,0)JSR(MotorStatusSUB,0)COP(TempMotor,S4A,1);
   172: COP(S4B,TempMotor,1)JSR(E300_StatusAlmWarnSUB,0)JSR(MotorStatusSUB,0)COP(TempMotor,S4B,1);
   173: COP(S5A,TempMotor,1)JSR(E300_StatusAlmWarnSUB,0)JSR(MotorStatusSUB,0)COP(TempMotor,S5A,1);
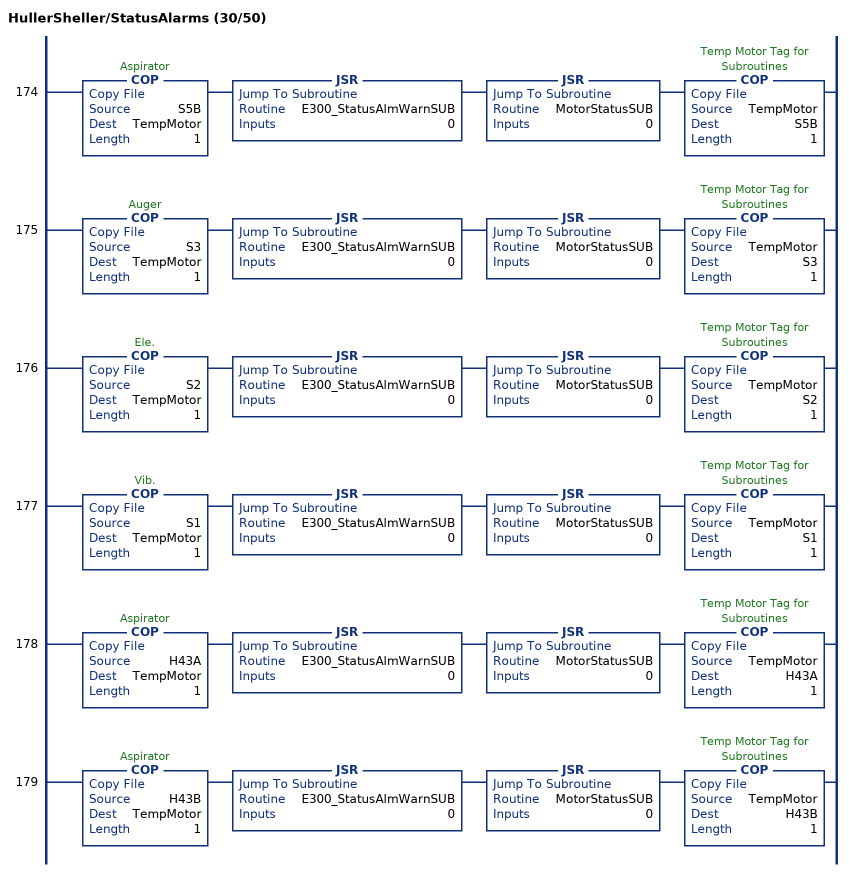
   174: COP(S5B,TempMotor,1)JSR(E300_StatusAlmWarnSUB,0)JSR(MotorStatusSUB,0)COP(TempMotor,S5B,1);
   175: COP(S3,TempMotor,1)JSR(E300_StatusAlmWarnSUB,0)JSR(MotorStatusSUB,0)COP(TempMotor,S3,1);
   176: COP(S2,TempMotor,1)JSR(E300_StatusAlmWarnSUB,0)JSR(MotorStatusSUB,0)COP(TempMotor,S2,1);
   177: COP(S1,TempMotor,1)JSR(E300_StatusAlmWarnSUB,0)JSR(MotorStatusSUB,0)COP(TempMotor,S1,1);
   178: COP(H43A,TempMotor,1)JSR(E300_StatusAlmWarnSUB,0)JSR(MotorStatusSUB,0)COP(TempMotor,H43A,1);
   179: COP(H43B,TempMotor,1)JSR(E300_StatusAlmWarnSUB,0)JSR(MotorStatusSUB,0)COP(TempMotor,H43B,1);
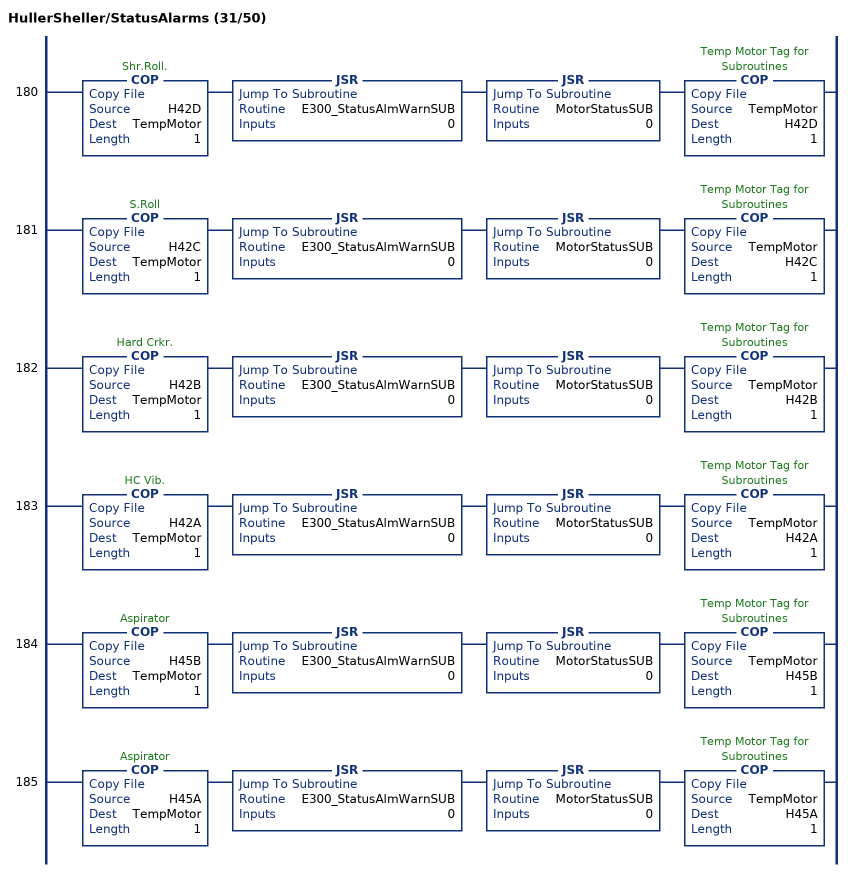
   180: COP(H42D,TempMotor,1)JSR(E300_StatusAlmWarnSUB,0)JSR(MotorStatusSUB,0)COP(TempMotor,H42D,1);
   181: COP(H42C,TempMotor,1)JSR(E300_StatusAlmWarnSUB,0)JSR(MotorStatusSUB,0)COP(TempMotor,H42C,1);
   182: COP(H42B,TempMotor,1)JSR(E300_StatusAlmWarnSUB,0)JSR(MotorStatusSUB,0)COP(TempMotor,H42B,1);
   183: COP(H42A,TempMotor,1)JSR(E300_StatusAlmWarnSUB,0)JSR(MotorStatusSUB,0)COP(TempMotor,H42A,1);
   184: COP(H45B,TempMotor,1)JSR(E300_StatusAlmWarnSUB,0)JSR(MotorStatusSUB,0)COP(TempMotor,H45B,1);
   185: COP(H45A,TempMotor,1)JSR(E300_StatusAlmWarnSUB,0)JSR(MotorStatusSUB,0)COP(TempMotor,H45A,1);
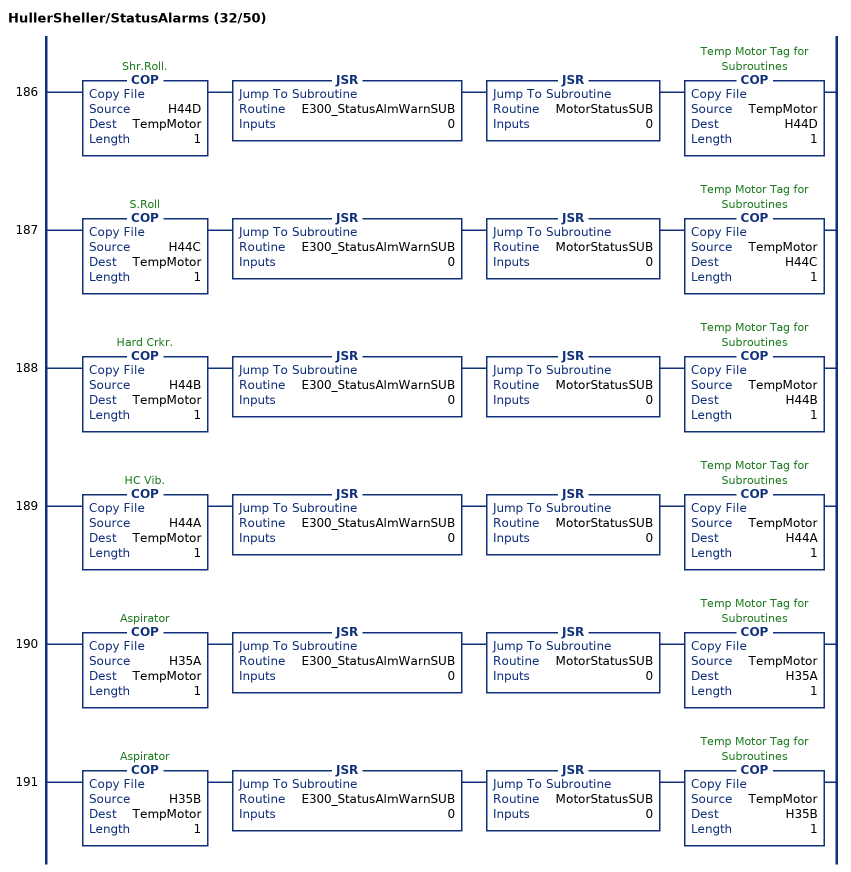
   186: COP(H44D,TempMotor,1)JSR(E300_StatusAlmWarnSUB,0)JSR(MotorStatusSUB,0)COP(TempMotor,H44D,1);
   187: COP(H44C,TempMotor,1)JSR(E300_StatusAlmWarnSUB,0)JSR(MotorStatusSUB,0)COP(TempMotor,H44C,1);
   188: COP(H44B,TempMotor,1)JSR(E300_StatusAlmWarnSUB,0)JSR(MotorStatusSUB,0)COP(TempMotor,H44B,1);
   189: COP(H44A,TempMotor,1)JSR(E300_StatusAlmWarnSUB,0)JSR(MotorStatusSUB,0)COP(TempMotor,H44A,1);
   190: COP(H35A,TempMotor,1)JSR(E300_StatusAlmWarnSUB,0)JSR(MotorStatusSUB,0)COP(TempMotor,H35A,1);
   191: COP(H35B,TempMotor,1)JSR(E300_StatusAlmWarnSUB,0)JSR(MotorStatusSUB,0)COP(TempMotor,H35B,1);
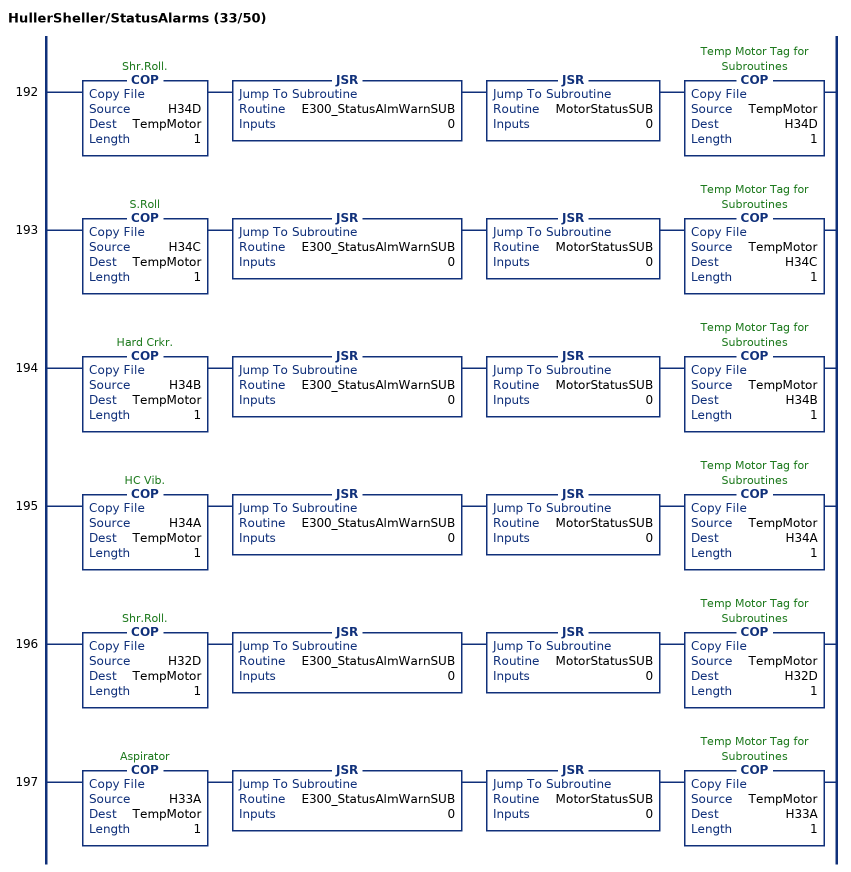
   192: COP(H34D,TempMotor,1)JSR(E300_StatusAlmWarnSUB,0)JSR(MotorStatusSUB,0)COP(TempMotor,H34D,1);
   193: COP(H34C,TempMotor,1)JSR(E300_StatusAlmWarnSUB,0)JSR(MotorStatusSUB,0)COP(TempMotor,H34C,1);
   194: COP(H34B,TempMotor,1)JSR(E300_StatusAlmWarnSUB,0)JSR(MotorStatusSUB,0)COP(TempMotor,H34B,1);
   195: COP(H34A,TempMotor,1)JSR(E300_StatusAlmWarnSUB,0)JSR(MotorStatusSUB,0)COP(TempMotor,H34A,1);
   196: COP(H32D,TempMotor,1)JSR(E300_StatusAlmWarnSUB,0)JSR(MotorStatusSUB,0)COP(TempMotor,H32D,1);
   197: COP(H33A,TempMotor,1)JSR(E300_StatusAlmWarnSUB,0)JSR(MotorStatusSUB,0)COP(TempMotor,H33A,1);
